Staubli VAL3: _kill.pgx

public program _kill()
  local string l_sMessage
begin
  // KILL KERNEL
  $jogPage(true)
  title("")
  cls()
  call language:message(l_sMessage,17)
  call use:timerDialog(l_sMessage,0)
  logMsg("[KERNEL] SUPERVISOR:Interface>Quit KERNEL")
  taskKill("Interface")
  taskKill("Point")
  taskKill("Remote")
  taskKill("Cycle")
  taskKill("Plc")
  taskKill("Action")
  watch(taskStatus("Interface")==-1,1)
  watch(taskStatus("Remote")==-1,1)
  watch(taskStatus("Cycle")==-1,1)
  watch(taskStatus("Plc")==-1,1)
  // save the last setting
  saveData:libSave()
  // save the cycle
  call processList:save()
  bQuit=false
  // give a time delay
  delay(1)
end
